# EPICS autosave request: tests/testfiles/cfg/SF_OpticsMCOR_PV.req
$(SYS):ONOFF
$(SYS):I-SET
